TYPE "PartCuttedBuffer_Item"
VERSION : 0.1
// Block: PartCuttedBuffer_Item
   STRUCT
      PTrkId : DInt;
      HeadCutPosition : LReal;
      TailCutPosition : LReal;
      R1_TailPosVirtPos : LReal;
      R2_TailPosVirtPos : LReal;
      Result : Int;
   END_STRUCT;

END_TYPE
